// TIA Portal V16 export
// export: Created 2023-03-31T06:57:52.9364437Z, ExportSetting WithDefaults, DisplayName Totally Integrated Automation Portal, DisplayVersion V16 Update 6, DisplayName TIA Portal Version Control Interface, DisplayVersion V16 Update 2, DisplayName TIA Portal Openness, DisplayVersion V16 Update 6, DisplayName STEP 7 Professional, DisplayVersion V16 Update 6, DisplayName STEP 7 Safety, DisplayVersion V16, DisplayName WinCC Advanced, DisplayVersion V16 Update 6
FUNCTION_BLOCK "EIT MNG"   // FB18, LAD
{ S7_Optimized_Access := 'FALSE' }
VERSION : 0.1
// EIT Management ver 0.0.1
// - Manage EIT Timer
// - Manage EIT Level memories
// stored: AutoNumber false, IsIECCheckEnabled false, SetENOAutomatically false, UDAEnableTagReadback false
   VAR DB_SPECIFIC
      Level : Struct
         _01 : Bool;   // "INTERNAL"
         _02 : Bool;   // "UPSTREAM"
         _03 : Bool;   // "DOWNSTREAM"
         _04 : Bool;   // "EXTERNAL"
         _05 : Bool;   // "OPERATOR"
         _06 : Bool;   // "AVAILABLE"
         _07 : Bool;   // "AVAILABLE"
         _08 : Bool;   // "AVAILABLE"
         _09 : Bool;   // "AVAILABLE"
         _10 : Bool;   // "BLOWER INTERNAL"
         _11 : Bool;   // "BLOWER UPSTREAM"
         _12 : Bool;   // "BLOWER DOWNSTREAM"
         _13 : Bool;   // "BLOWER EXTERNAL"
         _14 : Bool;   // "BLOWER OPERATOR"
         _15 : Bool;   // "BLOWER NO ALARMS ACTIVE"
         _16 : Bool;   // "NO ALARMS ACTIVE"
      END_STRUCT;
      Time_Level : Struct
         _01 : DInt;   // "INTERNAL"
         _02 : DInt;   // "UPSTREAM"
         _03 : DInt;   // "DOWNSTREAM"
         _04 : DInt;   // "EXTERNAL"
         _05 : DInt;   // "OPERATOR"
         _06 : DInt;   // "AVAILABLE"
         _07 : DInt;   // "AVAILABLE"
         _08 : DInt;   // "AVAILABLE"
         _09 : DInt;   // "AVAILABLE"
         _10 : DInt;   // "BLOWER INTERNAL"
         _11 : DInt;   // "BLOWER UPSTREAM"
         _12 : DInt;   // "BLOWER DOWNSTREAM"
         _13 : DInt;   // "BLOWER EXTERNAL"
         _14 : DInt;   // "BLOWER OPERATOR"
         _15 : DInt;   // "BLOWER NO ALARMS ACTIVE"
         _16 : DInt;   // "NO ALARMS ACTIVE"
      END_STRUCT;
      Times : Struct
         _01 : DInt;
         _02 : DInt;
         _03 : DInt;
         _04 : DInt;
         _05 : DInt;
         _06 : DInt;
         _07 : DInt;
         _08 : DInt;
         _09 : DInt;
         _10 : DInt;
         _11 : DInt;
         _12 : DInt;
         _13 : DInt;
         _14 : DInt;
         _15 : DInt;
         _16 : DInt;
      END_STRUCT;
   END_VAR
   VAR_TEMP
      RetVal : Int;
   END_VAR
   VAR_TEMP   // added for the SCL form of the ladder/FBD networks
      _w1 : Bool;
      _w2 : Bool;
   END_VAR
BEGIN

REGION Network 1: EIT - Reset memories - No alarms Active
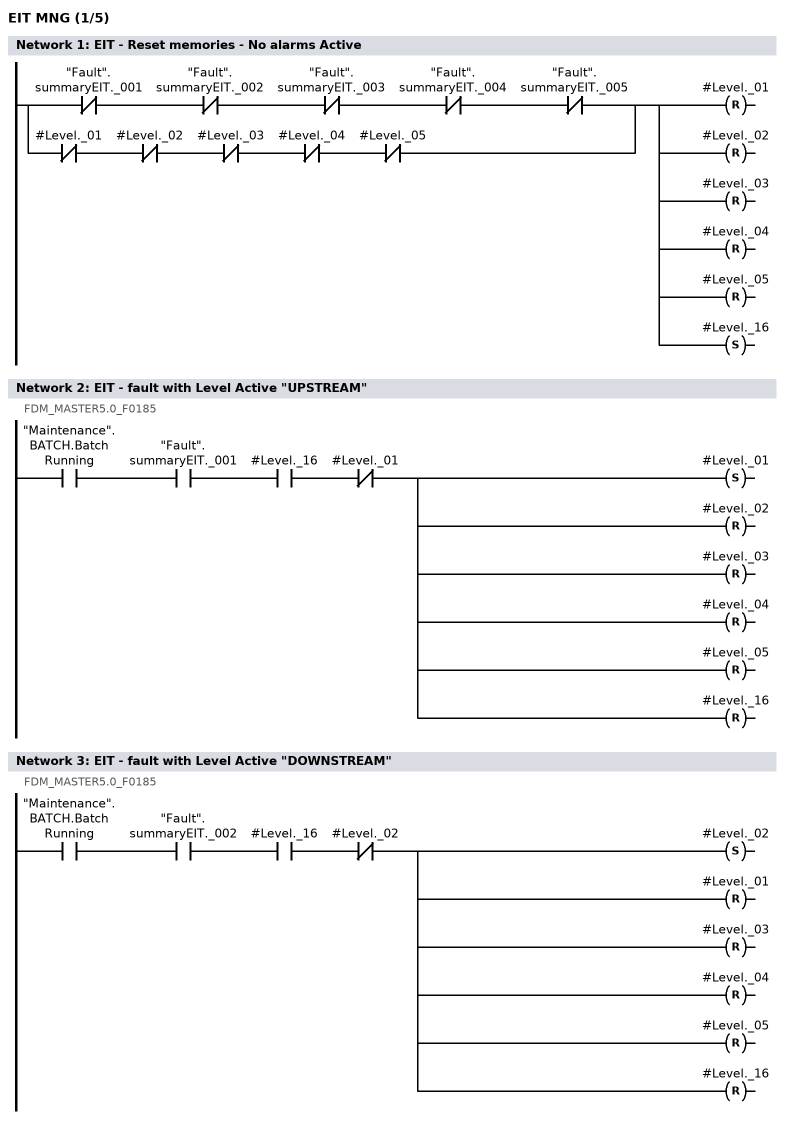
   RUNG wire#powerrail
      I_Contact( "Fault".summaryEIT._001 )
      I_Contact( "Fault".summaryEIT._002 )
      I_Contact( "Fault".summaryEIT._003 )
      I_Contact( "Fault".summaryEIT._004 )
      I_Contact( "Fault".summaryEIT._005 )
      wire#w1
      R_Coil( #Level._01 )
   END_RUNG
   RUNG wire#powerrail
      I_Contact( #Level._01 )
      I_Contact( #Level._02 )
      I_Contact( #Level._03 )
      I_Contact( #Level._04 )
      I_Contact( #Level._05 )
   END_RUNG wire#w1
   RUNG wire#w1
      R_Coil( #Level._02 )
   END_RUNG
   RUNG wire#w1
      R_Coil( #Level._03 )
   END_RUNG
   RUNG wire#w1
      R_Coil( #Level._04 )
   END_RUNG
   RUNG wire#w1
      R_Coil( #Level._05 )
   END_RUNG
   RUNG wire#w1
      S_Coil( #Level._16 )
   END_RUNG
   // the same network as SCL:
   #_w1 := (NOT "Fault".summaryEIT._001 AND NOT "Fault".summaryEIT._002 AND NOT "Fault".summaryEIT._003 AND NOT "Fault".summaryEIT._004 AND NOT "Fault".summaryEIT._005) OR (NOT #Level._01 AND NOT #Level._02 AND NOT #Level._03 AND NOT #Level._04 AND NOT #Level._05);
   IF #_w1 THEN
       #Level._01 := FALSE;
       #Level._02 := FALSE;
       #Level._03 := FALSE;
       #Level._04 := FALSE;
       #Level._05 := FALSE;
       #Level._16 := TRUE;
   END_IF;
END_REGION

REGION Network 2: EIT - fault with Level Active "UPSTREAM"
   // FDM_MASTER5.0_F0185
   RUNG wire#powerrail
      Contact( "Maintenance".BATCH.BatchRunning )
      Contact( "Fault".summaryEIT._001 )
      Contact( #Level._16 )
      I_Contact( #Level._01 )
      wire#w1
      S_Coil( #Level._01 )
   END_RUNG
   RUNG wire#w1
      R_Coil( #Level._02 )
   END_RUNG
   RUNG wire#w1
      R_Coil( #Level._03 )
   END_RUNG
   RUNG wire#w1
      R_Coil( #Level._04 )
   END_RUNG
   RUNG wire#w1
      R_Coil( #Level._05 )
   END_RUNG
   RUNG wire#w1
      R_Coil( #Level._16 )
   END_RUNG
   // the same network as SCL:
   #_w1 := "Maintenance".BATCH.BatchRunning AND "Fault".summaryEIT._001 AND #Level._16 AND NOT #Level._01;
   IF #_w1 THEN
       #Level._01 := TRUE;
       #Level._02 := FALSE;
       #Level._03 := FALSE;
       #Level._04 := FALSE;
       #Level._05 := FALSE;
       #Level._16 := FALSE;
   END_IF;
END_REGION

REGION Network 3: EIT - fault with Level Active "DOWNSTREAM"
   // FDM_MASTER5.0_F0185
   RUNG wire#powerrail
      Contact( "Maintenance".BATCH.BatchRunning )
      Contact( "Fault".summaryEIT._002 )
      Contact( #Level._16 )
      I_Contact( #Level._02 )
      wire#w1
      S_Coil( #Level._02 )
   END_RUNG
   RUNG wire#w1
      R_Coil( #Level._01 )
   END_RUNG
   RUNG wire#w1
      R_Coil( #Level._03 )
   END_RUNG
   RUNG wire#w1
      R_Coil( #Level._04 )
   END_RUNG
   RUNG wire#w1
      R_Coil( #Level._05 )
   END_RUNG
   RUNG wire#w1
      R_Coil( #Level._16 )
   END_RUNG
   // the same network as SCL:
   #_w1 := "Maintenance".BATCH.BatchRunning AND "Fault".summaryEIT._002 AND #Level._16 AND NOT #Level._02;
   IF #_w1 THEN
       #Level._02 := TRUE;
       #Level._01 := FALSE;
       #Level._03 := FALSE;
       #Level._04 := FALSE;
       #Level._05 := FALSE;
       #Level._16 := FALSE;
   END_IF;
END_REGION

REGION Network 4: EIT - fault with Level Active "EXTERNAL"
   // FDM_MASTER5.0_F0185
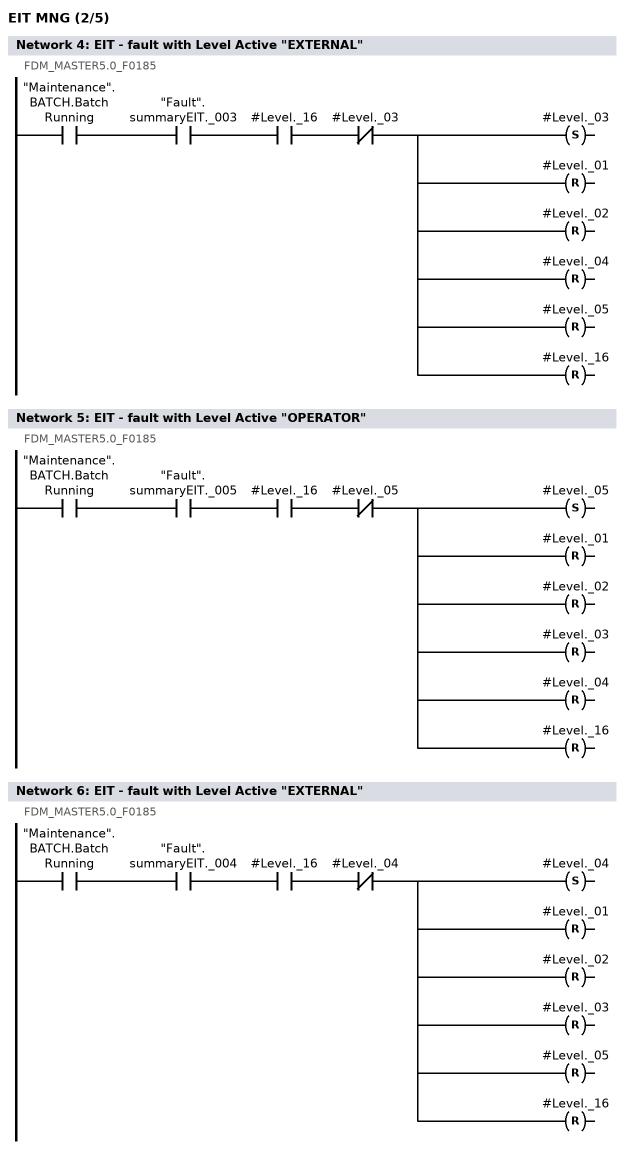
   RUNG wire#powerrail
      Contact( "Maintenance".BATCH.BatchRunning )
      Contact( "Fault".summaryEIT._003 )
      Contact( #Level._16 )
      I_Contact( #Level._03 )
      wire#w1
      S_Coil( #Level._03 )
   END_RUNG
   RUNG wire#w1
      R_Coil( #Level._01 )
   END_RUNG
   RUNG wire#w1
      R_Coil( #Level._02 )
   END_RUNG
   RUNG wire#w1
      R_Coil( #Level._04 )
   END_RUNG
   RUNG wire#w1
      R_Coil( #Level._05 )
   END_RUNG
   RUNG wire#w1
      R_Coil( #Level._16 )
   END_RUNG
   // the same network as SCL:
   #_w1 := "Maintenance".BATCH.BatchRunning AND "Fault".summaryEIT._003 AND #Level._16 AND NOT #Level._03;
   IF #_w1 THEN
       #Level._03 := TRUE;
       #Level._01 := FALSE;
       #Level._02 := FALSE;
       #Level._04 := FALSE;
       #Level._05 := FALSE;
       #Level._16 := FALSE;
   END_IF;
END_REGION

REGION Network 5: EIT - fault with Level Active "OPERATOR"
   // FDM_MASTER5.0_F0185
   RUNG wire#powerrail
      Contact( "Maintenance".BATCH.BatchRunning )
      Contact( "Fault".summaryEIT._005 )
      Contact( #Level._16 )
      I_Contact( #Level._05 )
      wire#w1
      S_Coil( #Level._05 )
   END_RUNG
   RUNG wire#w1
      R_Coil( #Level._01 )
   END_RUNG
   RUNG wire#w1
      R_Coil( #Level._02 )
   END_RUNG
   RUNG wire#w1
      R_Coil( #Level._03 )
   END_RUNG
   RUNG wire#w1
      R_Coil( #Level._04 )
   END_RUNG
   RUNG wire#w1
      R_Coil( #Level._16 )
   END_RUNG
   // the same network as SCL:
   #_w1 := "Maintenance".BATCH.BatchRunning AND "Fault".summaryEIT._005 AND #Level._16 AND NOT #Level._05;
   IF #_w1 THEN
       #Level._05 := TRUE;
       #Level._01 := FALSE;
       #Level._02 := FALSE;
       #Level._03 := FALSE;
       #Level._04 := FALSE;
       #Level._16 := FALSE;
   END_IF;
END_REGION

REGION Network 6: EIT - fault with Level Active "EXTERNAL"
   // FDM_MASTER5.0_F0185
   RUNG wire#powerrail
      Contact( "Maintenance".BATCH.BatchRunning )
      Contact( "Fault".summaryEIT._004 )
      Contact( #Level._16 )
      I_Contact( #Level._04 )
      wire#w1
      S_Coil( #Level._04 )
   END_RUNG
   RUNG wire#w1
      R_Coil( #Level._01 )
   END_RUNG
   RUNG wire#w1
      R_Coil( #Level._02 )
   END_RUNG
   RUNG wire#w1
      R_Coil( #Level._03 )
   END_RUNG
   RUNG wire#w1
      R_Coil( #Level._05 )
   END_RUNG
   RUNG wire#w1
      R_Coil( #Level._16 )
   END_RUNG
   // the same network as SCL:
   #_w1 := "Maintenance".BATCH.BatchRunning AND "Fault".summaryEIT._004 AND #Level._16 AND NOT #Level._04;
   IF #_w1 THEN
       #Level._04 := TRUE;
       #Level._01 := FALSE;
       #Level._02 := FALSE;
       #Level._03 := FALSE;
       #Level._05 := FALSE;
       #Level._16 := FALSE;
   END_IF;
END_REGION

REGION Network 7: Blower efficiency bits
   // FDM_MASTER5.0_F0185
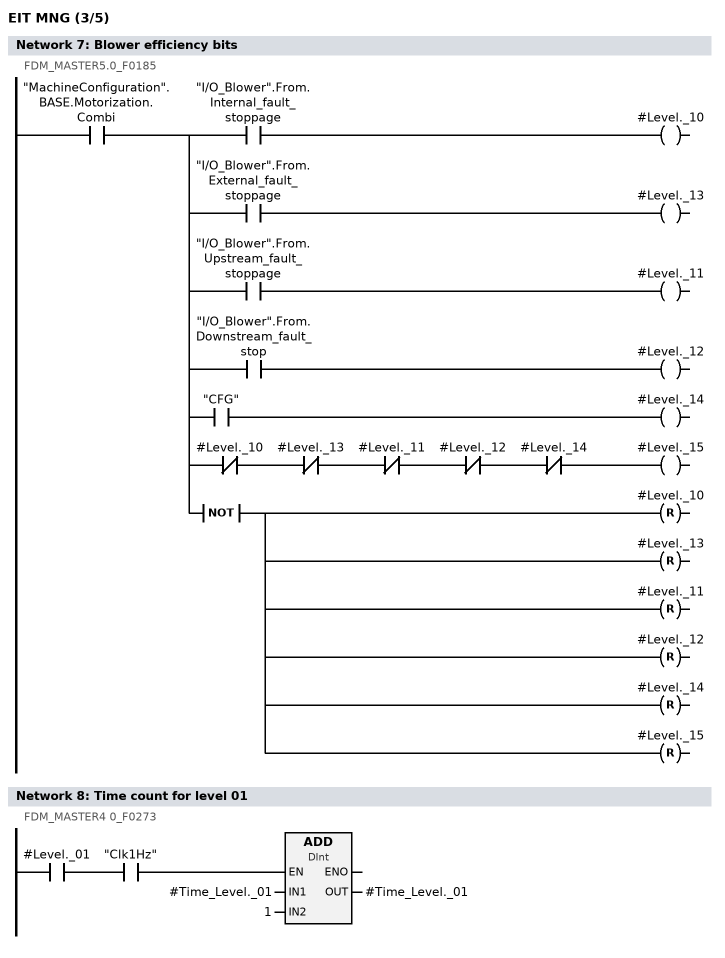
   RUNG wire#powerrail
      Contact( "MachineConfiguration".BASE.Motorization.Combi )
      wire#w1
      Contact( "I/O_Blower".From.Internal_fault_stoppage )
      Coil( #Level._10 )
   END_RUNG
   RUNG wire#w1
      Contact( "I/O_Blower".From.External_fault_stoppage )
      Coil( #Level._13 )
   END_RUNG
   RUNG wire#w1
      Contact( "I/O_Blower".From.Upstream_fault_stoppage )
      Coil( #Level._11 )
   END_RUNG
   RUNG wire#w1
      Contact( "I/O_Blower".From.Downstream_fault_stop )
      Coil( #Level._12 )
   END_RUNG
   RUNG wire#w1
      Contact( "CFG" )
      Coil( #Level._14 )
   END_RUNG
   RUNG wire#w1
      I_Contact( #Level._10 )
      I_Contact( #Level._13 )
      I_Contact( #Level._11 )
      I_Contact( #Level._12 )
      I_Contact( #Level._14 )
      Coil( #Level._15 )
   END_RUNG
   RUNG wire#w1
      Not()
      wire#w2
      R_Coil( #Level._10 )
   END_RUNG
   RUNG wire#w2
      R_Coil( #Level._13 )
   END_RUNG
   RUNG wire#w2
      R_Coil( #Level._11 )
   END_RUNG
   RUNG wire#w2
      R_Coil( #Level._12 )
   END_RUNG
   RUNG wire#w2
      R_Coil( #Level._14 )
   END_RUNG
   RUNG wire#w2
      R_Coil( #Level._15 )
   END_RUNG
   // the same network as SCL:
   #Level._10 := "MachineConfiguration".BASE.Motorization.Combi AND "I/O_Blower".From.Internal_fault_stoppage;
   #Level._13 := "MachineConfiguration".BASE.Motorization.Combi AND "I/O_Blower".From.External_fault_stoppage;
   #Level._11 := "MachineConfiguration".BASE.Motorization.Combi AND "I/O_Blower".From.Upstream_fault_stoppage;
   #Level._12 := "MachineConfiguration".BASE.Motorization.Combi AND "I/O_Blower".From.Downstream_fault_stop;
   #Level._14 := "MachineConfiguration".BASE.Motorization.Combi AND "CFG";
   #Level._15 := "MachineConfiguration".BASE.Motorization.Combi AND NOT #Level._10 AND NOT #Level._13 AND NOT #Level._11 AND NOT #Level._12 AND NOT #Level._14;
   IF NOT "MachineConfiguration".BASE.Motorization.Combi THEN
       #Level._10 := FALSE;
       #Level._13 := FALSE;
       #Level._11 := FALSE;
       #Level._12 := FALSE;
       #Level._14 := FALSE;
       #Level._15 := FALSE;
   END_IF;
END_REGION

REGION Network 8: Time count for level 01
   // FDM_MASTER4 0_F0273
   RUNG wire#powerrail
      Contact( #Level._01 )
      Contact( "Clk1Hz" )
      { S7_Templates := "SrcType := DInt"; S7_GenerateENO := "TRUE" } Add(in1 := #Time_Level._01, in2 := 1, out => #Time_Level._01)
   END_RUNG
   // the same network as SCL:
   IF #Level._01 AND "Clk1Hz" THEN #Time_Level._01 := #Time_Level._01 + 1; END_IF;
END_REGION

REGION Network 9: Time count for level 02
   // FDM_MASTER4 0_F0273
   // FDM_MASTER5.0_F0185
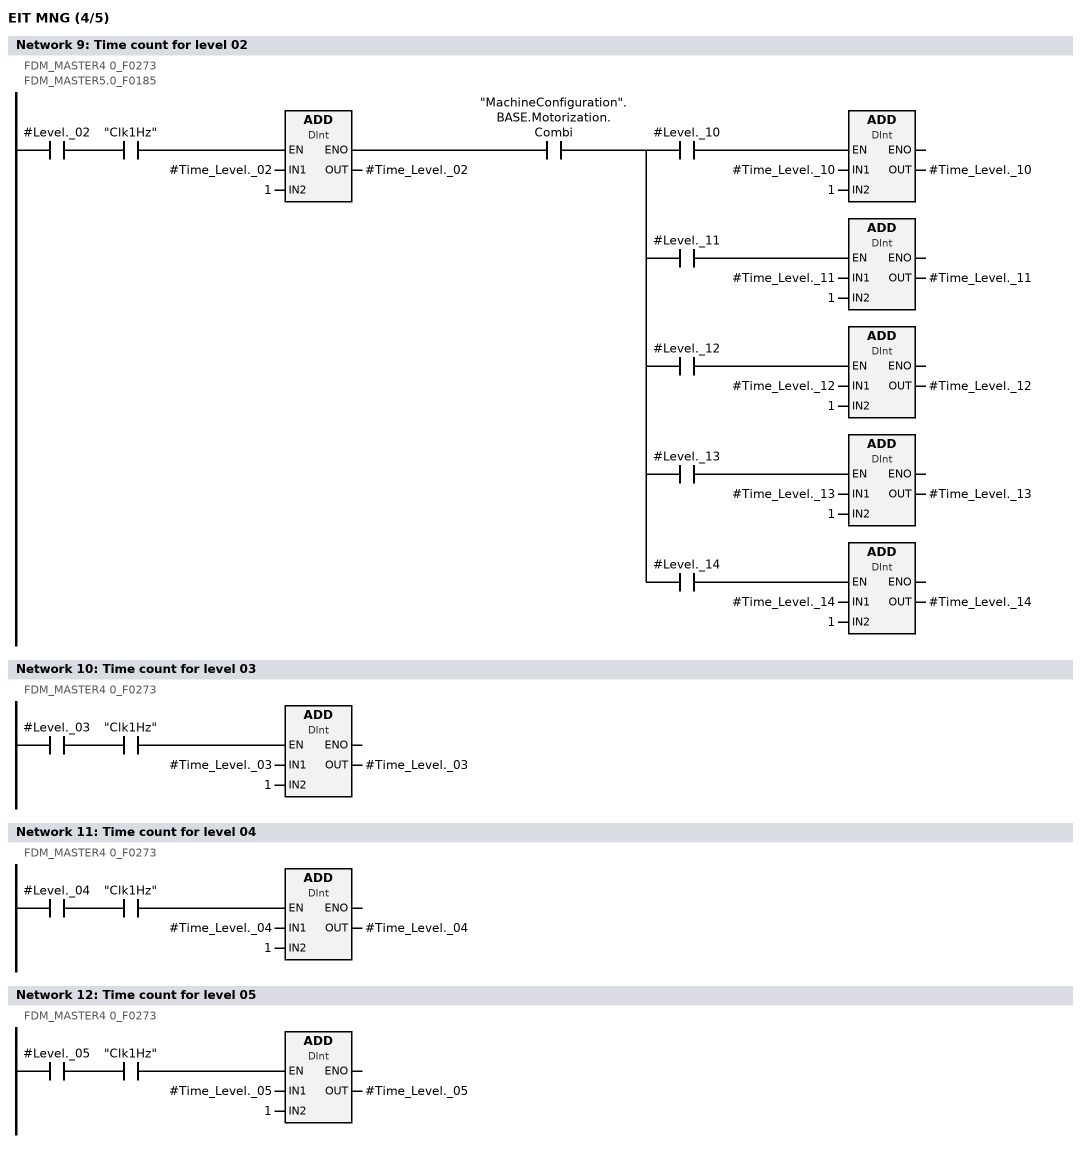
   RUNG wire#powerrail
      Contact( #Level._02 )
      Contact( "Clk1Hz" )
      { S7_Templates := "SrcType := DInt"; S7_GenerateENO := "TRUE" } Add(in1 := #Time_Level._02, in2 := 1, out => #Time_Level._02)
      Contact( "MachineConfiguration".BASE.Motorization.Combi )
      wire#w1
      Contact( #Level._10 )
      { S7_Templates := "SrcType := DInt"; S7_GenerateENO := "TRUE" } Add(in1 := #Time_Level._10, in2 := 1, out => #Time_Level._10)
   END_RUNG
   RUNG wire#w1
      Contact( #Level._11 )
      { S7_Templates := "SrcType := DInt"; S7_GenerateENO := "TRUE" } Add(in1 := #Time_Level._11, in2 := 1, out => #Time_Level._11)
   END_RUNG
   RUNG wire#w1
      Contact( #Level._12 )
      { S7_Templates := "SrcType := DInt"; S7_GenerateENO := "TRUE" } Add(in1 := #Time_Level._12, in2 := 1, out => #Time_Level._12)
   END_RUNG
   RUNG wire#w1
      Contact( #Level._13 )
      { S7_Templates := "SrcType := DInt"; S7_GenerateENO := "TRUE" } Add(in1 := #Time_Level._13, in2 := 1, out => #Time_Level._13)
   END_RUNG
   RUNG wire#w1
      Contact( #Level._14 )
      { S7_Templates := "SrcType := DInt"; S7_GenerateENO := "TRUE" } Add(in1 := #Time_Level._14, in2 := 1, out => #Time_Level._14)
   END_RUNG
   // the same network as SCL:
   // ENO of a box is taken as its EN; it also drops when the box reports an error
   #_w1 := #Level._02 AND "Clk1Hz";
   IF #_w1 THEN #Time_Level._02 := #Time_Level._02 + 1; END_IF;
   #_w2 := #_w1 AND "MachineConfiguration".BASE.Motorization.Combi;
   IF #_w2 AND #Level._10 THEN #Time_Level._10 := #Time_Level._10 + 1; END_IF;
   IF #_w2 AND #Level._11 THEN #Time_Level._11 := #Time_Level._11 + 1; END_IF;
   IF #_w2 AND #Level._12 THEN #Time_Level._12 := #Time_Level._12 + 1; END_IF;
   IF #_w2 AND #Level._13 THEN #Time_Level._13 := #Time_Level._13 + 1; END_IF;
   IF #_w2 AND #Level._14 THEN #Time_Level._14 := #Time_Level._14 + 1; END_IF;
END_REGION

REGION Network 10: Time count for level 03
   // FDM_MASTER4 0_F0273
   RUNG wire#powerrail
      Contact( #Level._03 )
      Contact( "Clk1Hz" )
      { S7_Templates := "SrcType := DInt"; S7_GenerateENO := "TRUE" } Add(in1 := #Time_Level._03, in2 := 1, out => #Time_Level._03)
   END_RUNG
   // the same network as SCL:
   IF #Level._03 AND "Clk1Hz" THEN #Time_Level._03 := #Time_Level._03 + 1; END_IF;
END_REGION

REGION Network 11: Time count for level 04
   // FDM_MASTER4 0_F0273
   RUNG wire#powerrail
      Contact( #Level._04 )
      Contact( "Clk1Hz" )
      { S7_Templates := "SrcType := DInt"; S7_GenerateENO := "TRUE" } Add(in1 := #Time_Level._04, in2 := 1, out => #Time_Level._04)
   END_RUNG
   // the same network as SCL:
   IF #Level._04 AND "Clk1Hz" THEN #Time_Level._04 := #Time_Level._04 + 1; END_IF;
END_REGION

REGION Network 12: Time count for level 05
   // FDM_MASTER4 0_F0273
   RUNG wire#powerrail
      Contact( #Level._05 )
      Contact( "Clk1Hz" )
      { S7_Templates := "SrcType := DInt"; S7_GenerateENO := "TRUE" } Add(in1 := #Time_Level._05, in2 := 1, out => #Time_Level._05)
   END_RUNG
   // the same network as SCL:
   IF #Level._05 AND "Clk1Hz" THEN #Time_Level._05 := #Time_Level._05 + 1; END_IF;
END_REGION

REGION Network 13: Time count for level 16 No alarm present
   // FDM_MASTER4 0_F0273
   // FDM_MASTER5.0_F0185
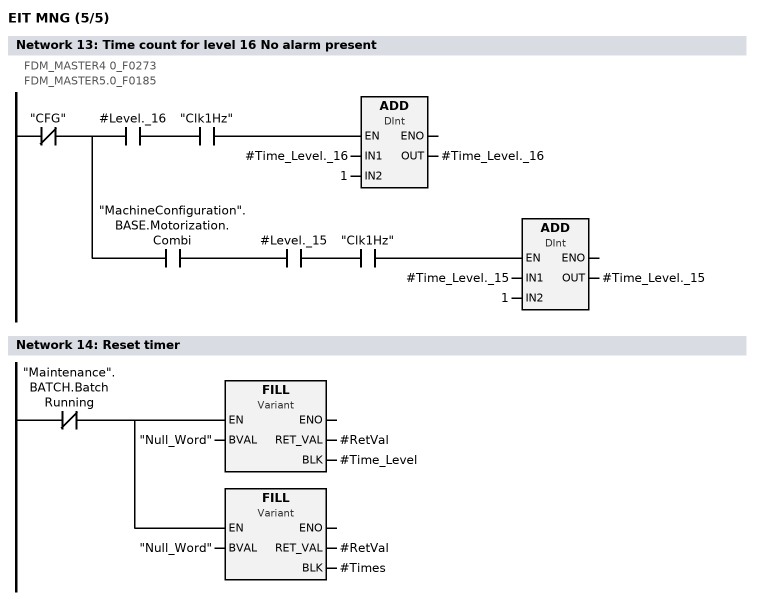
   RUNG wire#powerrail
      I_Contact( "CFG" )
      wire#w1
      Contact( #Level._16 )
      Contact( "Clk1Hz" )
      { S7_Templates := "SrcType := DInt"; S7_GenerateENO := "TRUE" } Add(in1 := #Time_Level._16, in2 := 1, out => #Time_Level._16)
   END_RUNG
   RUNG wire#w1
      Contact( "MachineConfiguration".BASE.Motorization.Combi )
      Contact( #Level._15 )
      Contact( "Clk1Hz" )
      { S7_Templates := "SrcType := DInt"; S7_GenerateENO := "TRUE" } Add(in1 := #Time_Level._15, in2 := 1, out => #Time_Level._15)
   END_RUNG
   // the same network as SCL:
   IF NOT "CFG" AND #Level._16 AND "Clk1Hz" THEN #Time_Level._16 := #Time_Level._16 + 1; END_IF;
   IF NOT "CFG" AND "MachineConfiguration".BASE.Motorization.Combi AND #Level._15 AND "Clk1Hz" THEN
       #Time_Level._15 := #Time_Level._15 + 1;
   END_IF;
END_REGION

REGION Network 14: Reset timer
   RUNG wire#powerrail
      I_Contact( "Maintenance".BATCH.BatchRunning )
      wire#w1
      { S7_Templates := "ptr_type := Variant" } FILL(BVAL := "Null_Word", RET_VAL => #RetVal, BLK => #Time_Level)
   END_RUNG
   RUNG wire#w1
      { S7_Templates := "ptr_type := Variant" } FILL(BVAL := "Null_Word", RET_VAL => #RetVal, BLK => #Times)
   END_RUNG
   // the same network as SCL:
   #_w1 := NOT "Maintenance".BATCH.BatchRunning;
   IF #_w1 THEN
       #RetVal := FILL(BVAL := "Null_Word", BLK => #Time_Level);
       #RetVal := FILL(BVAL := "Null_Word", BLK => #Times);
   END_IF;
END_REGION

NETWORK
TITLE = 
      SET;
      SAVE;

END_FUNCTION_BLOCK
